// TIA Portal project "bai8" (V15)

(* hardware
DEVICE "S7-1200 station_1"  S7-1200 Station
   slot 0: "Rack_0"  S7-1200 Rack  Rack  V1.0
   slot 1: "PLC_1"  CPU 1212C AC/DC/Rly  6ES7 212-1BE40-0XB0  V4.2
*)

// ===== PLC "PLC_1"  CPU 1212C AC/DC/Rly =====

VAR_GLOBAL   // PLC tag table "Default tag table"
   "Start" AT %M2.0 : Bool;
   "Stop" AT %M2.1 : Bool;
   "ON1" AT %Q0.0 : Bool;
   "Motor1" AT %Q0.1 : Bool;
   "Motor2" AT %Q0.2 : Bool;
   "Motor3" AT %Q0.3 : Bool;
   "Reset after error" AT %M2.3 : Bool;
   "stopall" AT %M0.0 : Bool;
END_VAR

// folder: System blocks/Program resources

DATA_BLOCK "IEC_Timer_0_DB"   // DB1
{ S7_Optimized_Access := 'TRUE' }
AUTHOR : Simatic
FAMILY : IEC
NAME : IEC_TMR
VERSION : 1.0
// stored: InstanceOfName IEC_TIMER
"IEC_TIMER"
BEGIN
END_DATA_BLOCK

DATA_BLOCK "IEC_Timer_0_DB1"   // DB2
{ S7_Optimized_Access := 'TRUE' }
AUTHOR : Simatic
FAMILY : IEC
NAME : IEC_TMR
VERSION : 1.0
// stored: InstanceOfName IEC_TIMER
"IEC_TIMER"
BEGIN
END_DATA_BLOCK

DATA_BLOCK "IEC_Timer_0_DB_2"   // DB4
{ S7_Optimized_Access := 'TRUE' }
AUTHOR : Simatic
FAMILY : IEC
NAME : IEC_TMR
VERSION : 1.0
// stored: InstanceOfName IEC_TIMER
"IEC_TIMER"
BEGIN
END_DATA_BLOCK

DATA_BLOCK "IEC_Timer_0_DB_3"   // DB5
{ S7_Optimized_Access := 'TRUE' }
AUTHOR : Simatic
FAMILY : IEC
NAME : IEC_TMR
VERSION : 1.0
// stored: InstanceOfName IEC_TIMER
"IEC_TIMER"
BEGIN
END_DATA_BLOCK

// folder: (top level)

ORGANIZATION_BLOCK "Main"   // OB1, LAD, ProgramCycle
TITLE = "Main Program Sweep (Cycle)"
{ S7_Optimized_Access := 'TRUE' }
VERSION : 0.1
   VAR_INPUT
      Initial_Call : Bool;   // Initial call of this OB
      Remanence : Bool;   // =True, if remanent data are available
   END_VAR
   VAR_TEMP   // added for the SCL form of the ladder/FBD networks
      _w1 : Bool;
   END_VAR
BEGIN

REGION Network 1
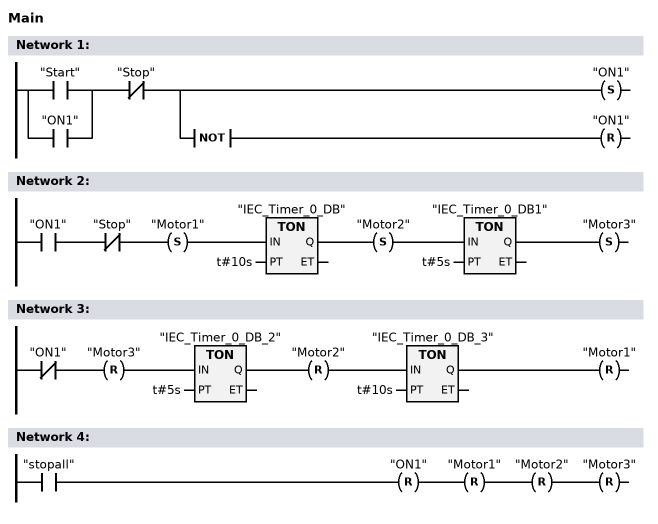
   RUNG wire#powerrail
      Contact( "Start" )
      wire#w1
      I_Contact( "Stop" )
      wire#w2
      S_Coil( "ON1" )
   END_RUNG
   RUNG wire#powerrail
      Contact( "ON1" )
   END_RUNG wire#w1
   RUNG wire#w2
      Not()
      R_Coil( "ON1" )
   END_RUNG
   // the same network as SCL:
   #_w1 := ("Start" OR "ON1") AND NOT "Stop";
   IF #_w1 THEN "ON1" := TRUE; END_IF;
   IF NOT #_w1 THEN "ON1" := FALSE; END_IF;
END_REGION

REGION Network 2
   #_w1 := "ON1" AND NOT "Stop";
   IF #_w1 THEN "Motor1" := TRUE; END_IF;
   "IEC_Timer_0_DB".TON(IN := #_w1, PT := t#10s);
   IF "IEC_Timer_0_DB".Q THEN "Motor2" := TRUE; END_IF;
   "IEC_Timer_0_DB1".TON(IN := "IEC_Timer_0_DB".Q, PT := t#5s);
   IF "IEC_Timer_0_DB1".Q THEN "Motor3" := TRUE; END_IF;
END_REGION

REGION Network 3
   IF NOT "ON1" THEN "Motor3" := FALSE; END_IF;
   "IEC_Timer_0_DB_2".TON(IN := NOT "ON1", PT := t#5s);
   IF "IEC_Timer_0_DB_2".Q THEN "Motor2" := FALSE; END_IF;
   "IEC_Timer_0_DB_3".TON(IN := "IEC_Timer_0_DB_2".Q, PT := t#10s);
   IF "IEC_Timer_0_DB_3".Q THEN "Motor1" := FALSE; END_IF;
END_REGION

REGION Network 4
   RUNG wire#powerrail
      Contact( "stopall" )
      R_Coil( "ON1" )
      R_Coil( "Motor1" )
      R_Coil( "Motor2" )
      R_Coil( "Motor3" )
   END_RUNG
   // the same network as SCL:
   IF "stopall" THEN
       "ON1" := FALSE;
       "Motor1" := FALSE;
       "Motor2" := FALSE;
       "Motor3" := FALSE;
   END_IF;
END_REGION
END_ORGANIZATION_BLOCK